(* CODESYS project WaterGASFC.export

Project tree, tasks and I/O mapping:
  function block Water_GA [SFC]: _aEmptying_active, _aEmptying_exit, _aEnd_active, _aEnd_exit, _aFilling_active, _aFilling_exit, _aInit_active, _aReady_active, _aReady_exit, _aWaterLvlCheck_active
*)

// Water_GA
FUNCTION_BLOCK Water_GA
VAR_INPUT
	(*Variabili d'ingresso esterne*)
	Do_: BOOL;					(* Variabile DO del GA Water*)
	DoWhat: Do_WaterWhat;		(* Variabile doWhat del GA Water*)
	WMFull: INT;				(* Valore indicativo di un cestello riempito d'acqua*)
	WMEmpty: INT;				(* Valore indicativo di un cestello svuotato dall'acqua*)
	LoWaterLvl: INT;			(* Valore indicativo di un cestello con piccola quantità d'acqua il cui sportello può essere aperto*)
	
	(*Variabili d'ingresso interne*)
	WaterLevel: INT;			(* Variabile d'aggancio al sensore di livello dell'acqua nel cestello*)
END_VAR
VAR_OUTPUT
	(* Variabili d'uscita esterne (ovvero verso l'alto, ovvero verso l'Automa di Politica*)	
	State: GA_STATE;			(* Variabile di stato del GA Water*)
	Done: BOOL;					(* Variabile DONE del GA Water*)
	NOwater: BOOL;				(* Variabile indicativa di un cestello privo d'acqua*)
	LoWater: BOOL;				(* Variabile indicativa di un cestello con una piccola quantità d'acqua al punto da poter aprire lo sportello senza conseguenze*)
	
	(*Variabili d'uscita interne*)
	ActFilling: BOOL;			(* Variabile d'aggancio verso l'attuatore ON/OFF di immissione dell'acqua*)
	ActEmptying: BOOL;			(* Variabile d'aggancio verso l'attuatore ON/OFF di scarico dell'acqua*)
	
END_VAR
VAR
END_VAR

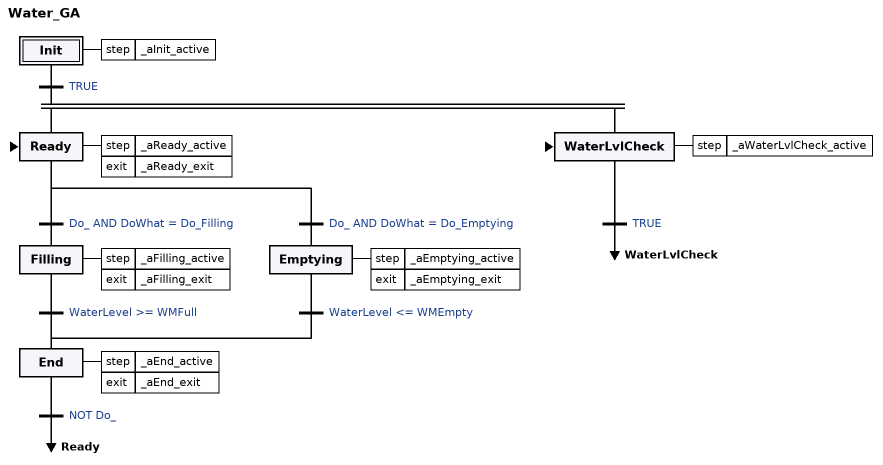
INITIAL_STEP Init:
    _aInit_active(N);  // step action
END_STEP
TRANSITION FROM Init TO (Ready, WaterLvlCheck)
    := TRUE;
END_TRANSITION
STEP Ready:
    _aReady_active(N);  // step action
    _aReady_exit(P0);  // exit action
END_STEP
STEP WaterLvlCheck:
    _aWaterLvlCheck_active(N);  // step action
END_STEP
TRANSITION FROM WaterLvlCheck TO WaterLvlCheck
    := TRUE;
END_TRANSITION
TRANSITION FROM Ready TO Filling
    := Do_ AND DoWhat = Do_Filling;
END_TRANSITION
STEP Filling:
    _aFilling_active(N);  // step action
    _aFilling_exit(P0);  // exit action
END_STEP
TRANSITION FROM Filling TO End
    := WaterLevel >= WMFull;
END_TRANSITION
TRANSITION FROM Ready TO Emptying
    := Do_ AND DoWhat = Do_Emptying;
END_TRANSITION
STEP Emptying:
    _aEmptying_active(N);  // step action
    _aEmptying_exit(P0);  // exit action
END_STEP
TRANSITION FROM Emptying TO End
    := WaterLevel <= WMEmpty;
END_TRANSITION
STEP End:
    _aEnd_active(N);  // step action
    _aEnd_exit(P0);  // exit action
END_STEP
TRANSITION FROM End TO Ready
    := NOT Do_;
END_TRANSITION

ACTION _aEmptying_active:
State := S_Busy;
ActEmptying := TRUE;
END_ACTION

ACTION _aEmptying_exit:
ActEmptying := FALSE;
END_ACTION

ACTION _aEnd_active:
Done := TRUE;
END_ACTION

ACTION _aEnd_exit:
Done := FALSE;
END_ACTION

ACTION _aFilling_active:
State := S_Busy;
ActFilling := TRUE;
END_ACTION

ACTION _aFilling_exit:
ActFilling := FALSE;
END_ACTION

ACTION _aInit_active:
State := S_Init;
END_ACTION

ACTION _aReady_active:
State := S_Ready;
END_ACTION

ACTION _aReady_exit:
State := S_Busy;
END_ACTION

ACTION _aWaterLvlCheck_active:
NOwater := WaterLevel <= WMEmpty;
IF NOwater THEN
	LoWater := TRUE;
ELSE
	LoWater := waterLevel <= LoWaterLvl;	
END_IF
END_ACTION

END_FUNCTION_BLOCK
